{attribute 'linkalways'} 
{attribute 'no_explicit_call' := 'This FB is a CLASS and must be accessed using methods or properties'}
{attribute 'enable_dynamic_creation'}
FUNCTION_BLOCK _SINT EXTENDS NumericDatatypeBase
VAR
	localData : SINT;
	activeData : REFERENCE TO SINT REF= localData;
END_VAR

PROPERTY PUBLIC Address : PVOID
GET
Address := ADR(activeData);
END_GET
END_PROPERTY

METHOD PUBLIC ClearReference
VAR_INPUT
END_VAR
activeData REF= localData;
END_METHOD

METHOD PUBLIC Clone : I_Datatype
VAR
    pClone : POINTER TO _SINT;
END_VAR
pClone := __NEW(_SINT(InitialValue := Value));
Clone := pClone^;
END_METHOD

METHOD FB_init : BOOL
VAR_INPUT
	bInitRetains : BOOL; // if TRUE, the retain variables are initialized (warm start / cold start)
	bInCopyCode : BOOL;  // if TRUE, the instance afterwards gets moved into the copy code (online change)
	InitialValue : SINT;
END_VAR
localData := InitialValue;
END_METHOD

PROPERTY PUBLIC IsFloat : BOOL
GET
IsFloat := FALSE;
END_GET
END_PROPERTY

PROPERTY PUBLIC IsSigned : BOOL
GET
IsSigned := TRUE;
END_GET
END_PROPERTY

PROPERTY PUBLIC LowerBound : SINT
GET
LowerBound := DatatypeLimits.SINT_LOWER_LIMIT;
END_GET
END_PROPERTY

METHOD PUBLIC MakeReferenceTo
VAR_INPUT
	ReferenceTarget : REFERENCE TO SINT;
END_VAR
activeData REF= ReferenceTarget;
END_METHOD

PROPERTY PUBLIC Name : T_MAXSTRING
GET
Name := 'SINT';
END_GET
END_PROPERTY

METHOD PROTECTED SerializeLowerbound
VAR_INPUT
	Serializer : I_Serializer;
END_VAR
Serializer.AddSint(Lowerbound);
END_METHOD

METHOD PROTECTED SerializeUpperbound
VAR_INPUT
	Serializer : I_Serializer;
END_VAR
Serializer.AddSint(Upperbound);
END_METHOD

METHOD PUBLIC SerializeWith
VAR_INPUT
	Serializer : I_Serializer;
END_VAR
Serializer.AddSint(activeData);
END_METHOD

PROPERTY PUBLIC Size : UDINT
GET
Size := SIZEOF(activeData);
END_GET
END_PROPERTY

METHOD TryDeserializeFrom : BOOL
VAR_INPUT
	Deserializer : I_Deserializer;
	Feedback : I_DeserializerFeedback;
END_VAR
TryDeserializeFrom := Deserializer.TryGetSint(activeData, Feedback);
END_METHOD

METHOD TryMakeReferenceTo : BOOL
VAR_INPUT
	Target : I_Datatype;
END_VAR
VAR
	pTargetData : POINTER TO SINT;
END_VAR
IF NOT (Target.Name = Name) THEN
	RETURN;
END_IF

pTargetData := Target.Address;
activeData REF= pTargetData^;
TryMakeReferenceTo := TRUE;
END_METHOD

PROPERTY PUBLIC UpperBound : SINT
GET
UpperBound :=  DatatypeLimits.SINT_UPPER_LIMIT;
END_GET
END_PROPERTY

PROPERTY PUBLIC Value : SINT
GET
Value := activeData;
END_GET
SET
activeData := Value;
END_SET
END_PROPERTY

END_FUNCTION_BLOCK

(* stored: Version 1.1.0.1, ProductVersion 3.1.4024.12
   POU _SINT: Id {502e39ab-9e51-05e0-3f42-5c0213f80731}, SpecialFunc None
   Folder Constructor: Id {200e17d5-5e22-0cd4-2b01-bd966d3a24d7}
   Folder Protected: Id {0bef026e-3a5c-025f-0d99-3559c686db4b}
   Property Address: Id {0fde92f2-8641-0bd3-11be-907e85d2b38f}
   Get Get: Id {d4b4046b-af6f-05fd-1330-2015bc92c9ec}
   Method ClearReference: Id {9f74a110-e14d-0743-321a-6b138d95cbcf}
   Method Clone: Id {324a4a0f-c6c9-0320-2032-2e7c0a354814}
   Method FB_init: Id {a5a9255c-15b7-0241-232d-977d74d144ef}
   Property IsFloat: Id {676344fb-a87f-06c2-041c-1d8780acf529}
   Get Get: Id {9006802e-1aef-04f5-03c0-46ab04b89221}
   Property IsSigned: Id {307db2a1-6e02-0cd1-2bf6-719d42a03df1}
   Get Get: Id {0b917e1f-8da8-0331-2005-390ed013de66}
   Property LowerBound: Id {27e42da2-e116-0d5e-1223-69677c335c76}
   Get Get: Id {6811e3ad-c85a-0ff9-245f-226cf28d721e}
   Method MakeReferenceTo: Id {43a737b6-c598-0a81-0f63-cff57cd231ee}
   Property Name: Id {8c8bd5c6-a592-0001-322b-9b62907cea13}
   Get Get: Id {e89008bb-a6bf-0299-2eca-bd456f8bfd0b}
   Method SerializeLowerbound: Id {6f092a90-69cf-0d0d-2b1b-e9aeae800f36}
   Method SerializeUpperbound: Id {8cfd7bca-9e43-0a59-087a-53b07ab6827a}
   Method SerializeWith: Id {2ab9f70d-02be-092c-3a52-ff270bacac30}
   Property Size: Id {94e2434b-5de3-087b-176a-8d51e212d28b}
   Get Get: Id {fae27f64-d3ae-054d-14aa-20b4d43d2fb9}
   Method TryDeserializeFrom: Id {1ed218e1-dc0b-0d70-0f41-f88756790c06}
   Method TryMakeReferenceTo: Id {81f53243-1f25-0396-2a76-bf26651a7b39}
   Property UpperBound: Id {5496765f-cace-002f-35da-21d924cc9b33}
   Get Get: Id {10d8d093-542d-0cee-39e8-05c9407c10c3}
   Property Value: Id {f875e7e0-6b72-0b0d-155e-c9dc2db69d06}
   Get Get: Id {c022731d-0fae-00b6-3ec5-3c23329db8d0}
   Set Set: Id {135d9454-85b6-0d0c-23ea-61e46246e123} *)
